{attribute 'GeneratedUsingTerminal: EL6080-0000-0018'}
{attribute addProperty BoxType "EL6080-0000-0018"}
{attribute addProperty Id "StatusAT %I*UINT2"}
{attribute addProperty CRC "131312374"}
{attribute addProperty Size "2"}
TYPE Status_07D3AAF6 EXTENDS InputBase_8311D824 :
STRUCT
	{attribute addProperty Name "Status"}
	Status AT %I* : UINT;
END_STRUCT
END_TYPE

(* stored: Version 1.2.0.0, ProductVersion 3.1.4024.11
   DUT Status_07D3AAF6: Id {57ebf408-8abd-4eb3-9c65-4bd8946e7b88} *)
